// TwinCAT 3 PLC project PRG_B_BaseDecorator
// Title: B_BaseDecorate
// Company: RafalOS
// Author: Rafał Osajda
// ProjectVersion: 0.0.0.2
// ProgramVersion: 3.1.4024.0
// libraries:
//   B_Base, * (RafalOS)
//   Tc2_Standard, * (Beckhoff Automation GmbH)
//   Tc2_System, * (Beckhoff Automation GmbH)
//   Tc3_Module, * (Beckhoff Automation GmbH)
// project tree:
//   / PlcTask.TcTTO
//   POUs Compilation/ PRG_Compilation.TcPOU
//   POUs/A03_FB_BaseLoggerElementDecorator/ FB_BaseLoggerElementDecoratorParent.TcPOU, ITF_BaseLoggerElementDecoratorParent.TcIO
//   POUs/A04_FB_BaseComponentDecorator/ FB_BaseComponentDecoratorParent.TcPOU, ITF_BaseComponentDecoratorParent.TcIO
//   POUs/A05_FB_BaseControlElementDecorator/ FB_BaseControlElementDecoratorParent.TcPOU, ITF_BaseControlElementDecoratorParent.TcIO
//   POUs/A06_FB_BaseGroupElementDecorator/ FB_BaseGroupElementDecoratorParent.TcPOU, ITF_BaseGroupElementDecoratorParent.TcIO (not stored)
//   POUs/A07_FB_BaseTopElementDecorator/ FB_BaseTopElementDecoratorParent.TcPOU, ITF_BaseTopElementDecoratorParent.TcIO
// real-time tasks:
//   TASK PlcTask: cycle T#10ms, priority 20, ADS port 350

CONFIGURATION PRG_B_BaseDecorator
    RESOURCE PLC ON TwinCAT3
        TASK PlcTask(INTERVAL := T#10ms, PRIORITY := 20);
        PROGRAM PRG_Compilation WITH PlcTask : PRG_Compilation;
    END_RESOURCE
END_CONFIGURATION

// ---- POUs/A03_FB_BaseLoggerElementDecorator/ITF_BaseLoggerElementDecoratorParent.TcIO
INTERFACE ITF_BaseLoggerElementDecoratorParent EXTENDS ITF_BaseLoggerElement

END_INTERFACE

// ---- POUs/A04_FB_BaseComponentDecorator/ITF_BaseComponentDecoratorParent.TcIO
INTERFACE ITF_BaseComponentDecoratorParent EXTENDS ITF_BaseComponent

END_INTERFACE

// ---- POUs/A05_FB_BaseControlElementDecorator/ITF_BaseControlElementDecoratorParent.TcIO
INTERFACE ITF_BaseControlElementDecoratorParent EXTENDS ITF_BaseControlElement

END_INTERFACE

// ---- POUs/A07_FB_BaseTopElementDecorator/ITF_BaseTopElementDecoratorParent.TcIO
INTERFACE ITF_BaseTopElementDecoratorParent EXTENDS ITF_BaseTopElement

END_INTERFACE

// ---- POUs Compilation/PRG_Compilation.TcPOU
PROGRAM PRG_Compilation
VAR
	fbLoggerElement				: FB_BaseLoggerElement;
	fbLoggerElementDecorator	: FB_BaseLoggerElementDecoratorParent (fbToDecorate := fbLoggerElement);
END_VAR

END_PROGRAM

// ---- POUs/A03_FB_BaseLoggerElementDecorator/FB_BaseLoggerElementDecoratorParent.TcPOU
FUNCTION_BLOCK FB_BaseLoggerElementDecoratorParent IMPLEMENTS ITF_BaseLoggerElementDecoratorParent
VAR
	itfLoggerElement					: ITF_BaseLoggerElement;
END_VAR

(*			
	EVERDE sp. z o.o.
	Rafał Osajda		24.03.2025		TC 4024.66
	Definicja nowego zgłoszenia
*)
METHOD PUBLIC EventsDefinition : BOOL
EventsDefinition		:= THIS^.itfLoggerElement.EventsDefinition ();
END_METHOD

METHOD FB_init : BOOL
VAR_INPUT
	bInitRetains : BOOL; // if TRUE, the retain variables are initialized (warm start / cold start)
	bInCopyCode : BOOL;  // if TRUE, the instance afterwards gets moved into the copy code (online change)
	fbToDecorate		: ITF_DecoratedElement;
END_VAR
THIS^.itfLoggerElement	:= fbToDecorate.GetITFLoggerElement ();
END_METHOD

METHOD PUBLIC GetCode : STRING
VAR_INPUT
END_VAR
GetCode			:= THIS^.itfLoggerElement.GetCode ();
END_METHOD

METHOD PUBLIC GetID : UINT
VAR_INPUT
END_VAR
GetID		:= THIS^.itfLoggerElement.GetID ();
END_METHOD

METHOD PUBLIC GetIdentyfier : ST_BaseElementIdentifier
VAR_INPUT
END_VAR
GetIdentyfier		:= THIS^.itfLoggerElement.GetIdentyfier ();
END_METHOD

METHOD PUBLIC GetName : ST_BaseLabel
VAR_INPUT
END_VAR
GetName		:= THIS^.itfLoggerElement.GetName ();
END_METHOD

METHOD PUBLIC GetType : E_BaseElementType
VAR_INPUT
END_VAR
GetType		:= THIS^.itfLoggerElement.GetType ();
END_METHOD

METHOD PUBLIC SetCode
VAR_INPUT
	sCode							: STRING;
	sAdd							: STRING;
END_VAR
THIS^.itfLoggerElement.SetCode (sCode := sCode, sAdd := sAdd);
END_METHOD

(*			
	EVERDE sp. z o.o.
	Rafał Osajda		03.10.2025		TC 4024.66
	nadawanie unikalnych ID dla zdarzeń
*)
METHOD PUBLIC SetEventsIDs : UINT
VAR_INPUT
	uiNewID		: UINT;
END_VAR
SetEventsIDs		:= THIS^.itfLoggerElement.SetEventsIDs (uiNewID := uiNewID);
END_METHOD

METHOD PUBLIC SetID : UINT
VAR_INPUT
	uiID					: UINT;
END_VAR
SetID		:= THIS^.itfLoggerElement.SetID (uiID := uiID);
END_METHOD

METHOD PUBLIC SetName
VAR_INPUT
	stName				: ST_BaseLabel;
END_VAR
THIS^.itfLoggerElement.SetName (stName := stName);
END_METHOD

METHOD PUBLIC SetType
VAR_INPUT
	eType					: E_BaseElementType;
END_VAR
THIS^.itfLoggerElement.SetType (eType := eType);
END_METHOD

END_FUNCTION_BLOCK

// ---- POUs/A04_FB_BaseComponentDecorator/FB_BaseComponentDecoratorParent.TcPOU
FUNCTION_BLOCK FB_BaseComponentDecoratorParent EXTENDS FB_BaseLoggerElementDecoratorParent IMPLEMENTS ITF_BaseComponentDecoratorParent
VAR
	itfComponent				: ITF_BaseComponent;
END_VAR

(*			
	EVERDE sp. z o.o.
	Rafał Osajda		24.03.2025		TC 4024.66
	Definicja nowego zgłoszenia
*)
METHOD PUBLIC EventsDefinition : BOOL
EventsDefinition		:= THIS^.itfComponent.EventsDefinition ();
END_METHOD

(*			
	EVERDE sp. z o.o.
	Rafał Osajda		27.03.2025		TC 4024.66
	Obsluga bledow sprawdzanie czy jakis blad sie nei pojawil i ustawienie stanu lub wylaczenie
*)
METHOD PUBLIC ExecuteEveryCycle_Error
VAR_INPUT
END_VAR
THIS^.itfComponent.ExecuteEveryCycle_Error ();
END_METHOD

(*			
	EVERDE sp. z o.o.
	Rafał Osajda		27.03.2025		TC 4024.66
	Wywolanie co cykl operacji 
*)
METHOD PUBLIC ExecuteEveryCycle_Operation
VAR_INPUT
END_VAR
THIS^.itfComponent.ExecuteEveryCycle_Operation ();
END_METHOD

(*			
	EVERDE sp. z o.o.
	Rafał Osajda		27.03.2025		TC 4024.66
	Aktualizacja flag 
*)
METHOD PUBLIC ExecuteEveryCycle_Status
VAR_INST
END_VAR
THIS^.itfComponent.ExecuteEveryCycle_Status ();
END_METHOD

(*			
	EVERDE sp. z o.o.
	Rafał Osajda		27.03.2025		TC 4024.66
	Testowanie czy nei pojawil sie jakis rozkaz i uruchomienie odpowiednich operacji
*)
METHOD PUBLIC ExecuteEveryCycle_Test
VAR_INPUT
END_VAR
THIS^.itfComponent.ExecuteEveryCycle_Test ();
END_METHOD

METHOD FB_init : BOOL
VAR_INPUT
	bInitRetains : BOOL; // if TRUE, the retain variables are initialized (warm start / cold start)
	bInCopyCode : BOOL;  // if TRUE, the instance afterwards gets moved into the copy code (online change)
	fbToDecorate		: ITF_DecoratedElement;
END_VAR
THIS^.itfComponent		:= fbToDecorate.GetITFComponent ();
END_METHOD

(*			
	EVERDE sp. z o.o.
	Rafał Osajda		03.10.2025		TC 4024.66
	
*)
METHOD PUBLIC FirstCycle : BOOL
VAR_INPUT
END_VAR
FirstCycle				:= THIS^.itfComponent.FirstCycle ();
END_METHOD

METHOD PUBLIC GetCode : STRING
VAR_INPUT
END_VAR
GetCode			:= THIS^.itfComponent.GetCode ();
END_METHOD

METHOD PUBLIC GetID : UINT
VAR_INPUT
END_VAR
GetID		:= THIS^.itfComponent.GetID ();
END_METHOD

METHOD PUBLIC GetIdentyfier : ST_BaseElementIdentifier
VAR_INPUT
END_VAR
GetIdentyfier		:= THIS^.itfComponent.GetIdentyfier ();
END_METHOD

METHOD PUBLIC GetName : ST_BaseLabel
VAR_INPUT
END_VAR
GetName		:= THIS^.itfComponent.GetName ();
END_METHOD

METHOD PUBLIC GetType : E_BaseElementType
VAR_INPUT
END_VAR
GetType		:= THIS^.itfComponent.GetType ();
END_METHOD

METHOD PUBLIC IsValidCommonData : BOOL
VAR_INPUT
END_VAR
IsValidCommonData			:= THIS^.itfComponent.IsValidCommonData ();
END_METHOD

(*			
	EVERDE sp. z o.o.
	Rafał Osajda		07.10.2025		TC 4024.66
	Dodpisywanie się do listy logera
*)
METHOD PUBLIC JoinTheLogger : BOOL
VAR_INPUT
END_VAR
JoinTheLogger	:= THIS^.itfComponent.JoinTheLogger ();
END_METHOD

METHOD PUBLIC LinkCommonData : BOOL
VAR_INPUT
	stCommonData				: REFERENCE TO ST_BaseCommonData;
END_VAR
LinkCommonData			:= THIS^.itfComponent.LinkCommonData (stCommonData := stCommonData);
END_METHOD

(*			
	EVERDE sp. z o.o.
	Rafał Osajda		26.03.2025		TC 4024.66
	Zwraca wartość
*)
METHOD PUBLIC ParameterGetValue : REAL
VAR_INPUT
	uiNumber				: UINT;
END_VAR
ParameterGetValue			:= THIS^.itfComponent.ParameterGetValue (uiNumber := uiNumber);
END_METHOD

METHOD PUBLIC Reset : BOOL
VAR_INPUT
END_VAR
Reset	:= THIS^.itfComponent.Reset ();
END_METHOD

METHOD PUBLIC ResetGetBusy : BOOL
VAR_INPUT
END_VAR
ResetGetBusy		:= THIS^.itfComponent.ResetGetBusy ();
END_METHOD

METHOD PUBLIC ResetGetStatus : BOOL
VAR_INPUT
END_VAR
ResetGetStatus			:= THIS^.itfComponent.ResetGetStatus ();
END_METHOD

METHOD PUBLIC SetCode
VAR_INPUT
	sCode							: STRING;
	sAdd							: STRING;
END_VAR
THIS^.itfComponent.SetCode (sCode := sCode, sAdd := sAdd);
END_METHOD

(*			
	EVERDE sp. z o.o.
	Rafał Osajda		03.10.2025		TC 4024.66
	nadawanie unikalnych ID dla zdarzeń
*)
METHOD PUBLIC SetEventsIDs : UINT
VAR_INPUT
	uiNewID		: UINT;
END_VAR
SetEventsIDs		:= THIS^.itfComponent.SetEventsIDs (uiNewID := uiNewID);
END_METHOD

METHOD PUBLIC SetID : UINT
VAR_INPUT
	uiID					: UINT;
END_VAR
SetID		:= THIS^.itfComponent.SetID (uiID := uiID);
END_METHOD

METHOD PUBLIC SetName
VAR_INPUT
	stName				: ST_BaseLabel;
END_VAR
THIS^.itfComponent.SetName (stName := stName);
END_METHOD

METHOD PUBLIC SetType
VAR_INPUT
	eType					: E_BaseElementType;
END_VAR
THIS^.itfComponent.SetType (eType := eType);
END_METHOD

END_FUNCTION_BLOCK

// ---- POUs/A05_FB_BaseControlElementDecorator/FB_BaseControlElementDecoratorParent.TcPOU
FUNCTION_BLOCK FB_BaseControlElementDecoratorParent EXTENDS FB_BaseComponentDecoratorParent IMPLEMENTS ITF_BaseControlElementDecoratorParent
VAR
	itfControlElement				: ITF_BaseControlElement;
END_VAR

(*			
	EVERDE sp. z o.o.
	Rafał Osajda		24.03.2025		TC 4024.66
	Definicja nowego zgłoszenia
*)
METHOD PUBLIC EventsDefinition : BOOL
EventsDefinition		:= THIS^.itfControlElement.EventsDefinition ();
END_METHOD

(*			
	EVERDE sp. z o.o.
	Rafał Osajda		27.03.2025		TC 4024.66
	Obsluga bledow sprawdzanie czy jakis blad sie nei pojawil i ustawienie stanu lub wylaczenie
*)
METHOD PUBLIC ExecuteEveryCycle_Error
VAR_INPUT
END_VAR
THIS^.itfControlElement.ExecuteEveryCycle_Error ();
END_METHOD

(*			
	EVERDE sp. z o.o.
	Rafał Osajda		27.03.2025		TC 4024.66
	Wywolanie co cykl operacji 
*)
METHOD PUBLIC ExecuteEveryCycle_Operation
VAR_INPUT
END_VAR
THIS^.itfControlElement.ExecuteEveryCycle_Operation ();
END_METHOD

(*			
	EVERDE sp. z o.o.
	Rafał Osajda		27.03.2025		TC 4024.66
	Aktualizacja flag 
*)
METHOD PUBLIC ExecuteEveryCycle_Status
VAR_INST
END_VAR
THIS^.itfControlElement.ExecuteEveryCycle_Status ();
END_METHOD

(*			
	EVERDE sp. z o.o.
	Rafał Osajda		27.03.2025		TC 4024.66
	Testowanie czy nei pojawil sie jakis rozkaz i uruchomienie odpowiednich operacji
*)
METHOD PUBLIC ExecuteEveryCycle_Test
VAR_INPUT
END_VAR
THIS^.itfControlElement.ExecuteEveryCycle_Test ();
END_METHOD

METHOD FB_init : BOOL
VAR_INPUT
	bInitRetains : BOOL; // if TRUE, the retain variables are initialized (warm start / cold start)
	bInCopyCode : BOOL;  // if TRUE, the instance afterwards gets moved into the copy code (online change)
	fbToDecorate		: ITF_DecoratedElement;
END_VAR
THIS^.itfControlElement	:= fbToDecorate.GetITFControlElement ();
END_METHOD

(*			
	EVERDE sp. z o.o.
	Rafał Osajda		03.10.2025		TC 4024.66
	
*)
METHOD PUBLIC FirstCycle : BOOL
VAR_INPUT
END_VAR
FirstCycle				:= THIS^.itfControlElement.FirstCycle ();
END_METHOD

METHOD PUBLIC GetCode : STRING
VAR_INPUT
END_VAR
GetCode			:= THIS^.itfControlElement.GetCode ();
END_METHOD

(*			
	EVERDE sp. z o.o.
	Rafał Osajda		30.04.2025		TC 4024.66
	Zwraca czy element jest czymś zajety
*)
METHOD PUBLIC GetDoNothing : BOOL
GetDoNothing		:= THIS^.itfControlElement.GetDoNothing ();
END_METHOD

METHOD PUBLIC GetID : UINT
VAR_INPUT
END_VAR
GetID		:= THIS^.itfControlElement.GetID ();
END_METHOD

METHOD PUBLIC GetIdentyfier : ST_BaseElementIdentifier
VAR_INPUT
END_VAR
GetIdentyfier		:= THIS^.itfControlElement.GetIdentyfier ();
END_METHOD

METHOD PUBLIC GetName : ST_BaseLabel
VAR_INPUT
END_VAR
GetName		:= THIS^.itfControlElement.GetName ();
END_METHOD

(*			
	EVERDE sp. z o.o.
	Rafał Osajda		30.04.2025		TC 4024.66
	Zwraca czy element jest w pozycji 0 - referencyjnej
*)
METHOD PUBLIC GetPosition0 : BOOL
GetPosition0	:= THIS^.itfControlElement.GetPosition0 ();
END_METHOD

METHOD PUBLIC GetType : E_BaseElementType
VAR_INPUT
END_VAR
GetType		:= THIS^.itfControlElement.GetType ();
END_METHOD

(*			
	EVERDE sp. z o.o.
	Rafał Osajda		31.03.2025		TC 4024.66
	Flaga że w tej sesji pracy maszyny element został już wybazowany
*)
METHOD PUBLIC HomingGetDone : BOOL
VAR_INPUT
END_VAR
HomingGetDone	:= THIS^.itfControlElement.HomingGetDone ();
END_METHOD

(*			
	EVERDE sp. z o.o.
	Rafał Osajda		11.04.2025		TC 4024.66
	Zwraca czy bazowanie jest potrzebne
*)
METHOD PUBLIC HomingGetIsNeeded : BOOL
VAR_INPUT
END_VAR
HomingGetIsNeeded	:= THIS^.itfControlElement.HomingGetIsNeeded ();
END_METHOD

(*			
	EVERDE sp. z o.o.
	Rafał Osajda		27.05.2025		TC 4024.66
	Uruchomienie metody bazowania
*)
METHOD PUBLIC HomingStart
VAR_INPUT
END_VAR
THIS^.itfControlElement.HomingStart ();
END_METHOD

METHOD PUBLIC IsValidCommonData : BOOL
VAR_INPUT
END_VAR
IsValidCommonData			:= THIS^.itfControlElement.IsValidCommonData ();
END_METHOD

(*			
	EVERDE sp. z o.o.
	Rafał Osajda		07.10.2025		TC 4024.66
	Dodpisywanie się do listy logera
*)
METHOD PUBLIC JoinTheLogger : BOOL
VAR_INPUT
END_VAR
JoinTheLogger	:= THIS^.itfControlElement.JoinTheLogger ();
END_METHOD

METHOD PUBLIC LinkCommonData : BOOL
VAR_INPUT
	stCommonData				: REFERENCE TO ST_BaseCommonData;
END_VAR
LinkCommonData			:= THIS^.itfControlElement.LinkCommonData (stCommonData := stCommonData);
END_METHOD

METHOD PUBLIC LinkSS1 : BOOL
VAR_INPUT
	fbSS1			: ITF_BaseFlagGet;
END_VAR
LinkSS1		:= THIS^.itfControlElement.LinkSS1 (fbSS1 := fbSS1);
END_METHOD

METHOD PUBLIC LinkSTO : BOOL
VAR_INPUT
	fbSTO			: ITF_BaseFlagGet;
END_VAR
LinkSTO		:= THIS^.itfControlElement.LinkSTO (fbSTO := fbSTO);
END_METHOD

(*			
	EVERDE sp. z o.o.
	Rafał Osajda		31.03.2025		TC 4024.66
	Zwraca status zasilania	
*)
METHOD PUBLIC PowerGetStatus : BOOL
VAR_INPUT
END_VAR
PowerGetStatus		:= THIS^.itfControlElement.PowerGetStatus ();
END_METHOD

(*			
	EVERDE sp. z o.o.
	Rafał Osajda		31.03.2025		TC 4024.66
	Wyłączenie zasilania
*)
METHOD PUBLIC PowerTurnOff : BOOL
VAR_INPUT
END_VAR
PowerTurnOff		:= THIS^.itfControlElement.PowerTurnOff ();
END_METHOD

(*			
	EVERDE sp. z o.o.
	Rafał Osajda		31.03.2025		TC 4024.66
	Uruchomienie zasialania
*)
METHOD PUBLIC PowerTurnOn
VAR_INPUT
END_VAR
THIS^.itfControlElement.PowerTurnOn ();
END_METHOD

METHOD PUBLIC Reset : BOOL
VAR_INPUT
END_VAR
Reset	:= THIS^.itfControlElement.Reset ();
END_METHOD

METHOD PUBLIC ResetGetBusy : BOOL
VAR_INPUT
END_VAR
ResetGetBusy		:= THIS^.itfControlElement.ResetGetBusy ();
END_METHOD

METHOD PUBLIC ResetGetStatus : BOOL
VAR_INPUT
END_VAR
ResetGetStatus			:= THIS^.itfControlElement.ResetGetStatus ();
END_METHOD

METHOD PUBLIC SetCode
VAR_INPUT
	sCode							: STRING;
	sAdd							: STRING;
END_VAR
THIS^.itfControlElement.SetCode (sCode := sCode, sAdd := sAdd);
END_METHOD

(*			
	EVERDE sp. z o.o.
	Rafał Osajda		03.10.2025		TC 4024.66
	nadawanie unikalnych ID dla zdarzeń
*)
METHOD PUBLIC SetEventsIDs : UINT
VAR_INPUT
	uiNewID		: UINT;
END_VAR
SetEventsIDs		:= THIS^.itfControlElement.SetEventsIDs (uiNewID := uiNewID);
END_METHOD

METHOD PUBLIC SetID : UINT
VAR_INPUT
	uiID					: UINT;
END_VAR
SetID		:= THIS^.itfControlElement.SetID (uiID := uiID);
END_METHOD

METHOD PUBLIC SetName
VAR_INPUT
	stName				: ST_BaseLabel;
END_VAR
THIS^.itfControlElement.SetName (stName := stName);
END_METHOD

METHOD PUBLIC SetType
VAR_INPUT
	eType					: E_BaseElementType;
END_VAR
THIS^.itfControlElement.SetType (eType := eType);
END_METHOD

END_FUNCTION_BLOCK

// ---- POUs/A06_FB_BaseGroupElementDecorator/FB_BaseGroupElementDecoratorParent.TcPOU
FUNCTION_BLOCK FB_BaseGroupElementDecoratorParent EXTENDS FB_BaseControlElementDecoratorParent IMPLEMENTS ITF_BaseGroupElementDecoratorParent
VAR
	itfGroupElement				: ITF_BaseGroupElement;
END_VAR

(*			
	EVERDE sp. z o.o.
	Rafał Osajda		24.03.2025		TC 4024.66
	Definicja nowego zgłoszenia
*)
METHOD PUBLIC EventsDefinition : BOOL
EventsDefinition		:= THIS^.itfGroupElement.EventsDefinition ();
END_METHOD

(*			
	EVERDE sp. z o.o.
	Rafał Osajda		27.03.2025		TC 4024.66
	Obsluga bledow sprawdzanie czy jakis blad sie nei pojawil i ustawienie stanu lub wylaczenie
*)
METHOD PUBLIC ExecuteEveryCycle_Error
VAR_INPUT
END_VAR
THIS^.itfGroupElement.ExecuteEveryCycle_Error ();
END_METHOD

(*			
	EVERDE sp. z o.o.
	Rafał Osajda		27.03.2025		TC 4024.66
	Wywolanie co cykl operacji 
*)
METHOD PUBLIC ExecuteEveryCycle_Operation
VAR_INPUT
END_VAR
THIS^.itfGroupElement.ExecuteEveryCycle_Operation ();
END_METHOD

(*			
	EVERDE sp. z o.o.
	Rafał Osajda		27.03.2025		TC 4024.66
	Aktualizacja flag 
*)
METHOD PUBLIC ExecuteEveryCycle_Status
VAR_INST
END_VAR
THIS^.itfGroupElement.ExecuteEveryCycle_Status ();
END_METHOD

(*			
	EVERDE sp. z o.o.
	Rafał Osajda		27.03.2025		TC 4024.66
	Testowanie czy nei pojawil sie jakis rozkaz i uruchomienie odpowiednich operacji
*)
METHOD PUBLIC ExecuteEveryCycle_Test
VAR_INPUT
END_VAR
THIS^.itfGroupElement.ExecuteEveryCycle_Test ();
END_METHOD

METHOD FB_init : BOOL
VAR_INPUT
	bInitRetains : BOOL; // if TRUE, the retain variables are initialized (warm start / cold start)
	bInCopyCode : BOOL;  // if TRUE, the instance afterwards gets moved into the copy code (online change)
	fbToDecorate		: ITF_DecoratedElement;
END_VAR
THIS^.itfGroupElement	:= fbToDecorate.GetITFGroupElement ();
END_METHOD

(*			
	EVERDE sp. z o.o.
	Rafał Osajda		03.10.2025		TC 4024.66
	
*)
METHOD PUBLIC FirstCycle : BOOL
VAR_INPUT
END_VAR
FirstCycle				:= THIS^.itfGroupElement.FirstCycle ();
END_METHOD

METHOD PUBLIC GetCode : STRING
VAR_INPUT
END_VAR
GetCode			:= THIS^.itfGroupElement.GetCode ();
END_METHOD

(*			
	EVERDE sp. z o.o.
	Rafał Osajda		30.04.2025		TC 4024.66
	Zwraca czy element jest czymś zajety
*)
METHOD PUBLIC GetDoNothing : BOOL
GetDoNothing		:= THIS^.itfGroupElement.GetDoNothing ();
END_METHOD

METHOD PUBLIC GetID : UINT
VAR_INPUT
END_VAR
GetID		:= THIS^.itfGroupElement.GetID ();
END_METHOD

METHOD PUBLIC GetIdentyfier : ST_BaseElementIdentifier
VAR_INPUT
END_VAR
GetIdentyfier		:= THIS^.itfGroupElement.GetIdentyfier ();
END_METHOD

METHOD PUBLIC GetName : ST_BaseLabel
VAR_INPUT
END_VAR
GetName		:= THIS^.itfGroupElement.GetName ();
END_METHOD

(*			
	EVERDE sp. z o.o.
	Rafał Osajda		30.04.2025		TC 4024.66
	Zwraca czy element jest w pozycji 0 - referencyjnej
*)
METHOD PUBLIC GetPosition0 : BOOL
GetPosition0	:= THIS^.itfGroupElement.GetPosition0 ();
END_METHOD

METHOD PUBLIC GetType : E_BaseElementType
VAR_INPUT
END_VAR
GetType		:= THIS^.itfGroupElement.GetType ();
END_METHOD

(*			
	EVERDE sp. z o.o.
	Rafał Osajda		31.03.2025		TC 4024.66
	Flaga że w tej sesji pracy maszyny element został już wybazowany
*)
METHOD PUBLIC HomingGetDone : BOOL
VAR_INPUT
END_VAR
HomingGetDone	:= THIS^.itfGroupElement.HomingGetDone ();
END_METHOD

(*			
	EVERDE sp. z o.o.
	Rafał Osajda		11.04.2025		TC 4024.66
	Zwraca czy bazowanie jest potrzebne
*)
METHOD PUBLIC HomingGetIsNeeded : BOOL
VAR_INPUT
END_VAR
HomingGetIsNeeded	:= THIS^.itfGroupElement.HomingGetIsNeeded ();
END_METHOD

(*			
	EVERDE sp. z o.o.
	Rafał Osajda		27.05.2025		TC 4024.66
	Uruchomienie metody bazowania
*)
METHOD PUBLIC HomingStart
VAR_INPUT
END_VAR
THIS^.itfGroupElement.HomingStart ();
END_METHOD

METHOD PUBLIC IsValidCommonData : BOOL
VAR_INPUT
END_VAR
IsValidCommonData			:= THIS^.itfGroupElement.IsValidCommonData ();
END_METHOD

(*			
	EVERDE sp. z o.o.
	Rafał Osajda		07.10.2025		TC 4024.66
	Dodpisywanie się do listy logera
*)
METHOD PUBLIC JoinTheLogger : BOOL
VAR_INPUT
END_VAR
JoinTheLogger	:= THIS^.itfGroupElement.JoinTheLogger ();
END_METHOD

METHOD PUBLIC LinkCommonData : BOOL
VAR_INPUT
	stCommonData				: REFERENCE TO ST_BaseCommonData;
END_VAR
LinkCommonData			:= THIS^.itfGroupElement.LinkCommonData (stCommonData := stCommonData);
END_METHOD

METHOD PUBLIC LinkSS1 : BOOL
VAR_INPUT
	fbSS1			: ITF_BaseFlagGet;
END_VAR
LinkSS1		:= THIS^.itfGroupElement.LinkSS1 (fbSS1 := fbSS1);
END_METHOD

METHOD PUBLIC LinkSTO : BOOL
VAR_INPUT
	fbSTO			: ITF_BaseFlagGet;
END_VAR
LinkSTO		:= THIS^.itfGroupElement.LinkSTO (fbSTO := fbSTO);
END_METHOD

(*			
	EVERDE sp. z o.o.
	Rafał Osajda		31.03.2025		TC 4024.66
	Zwraca status zasilania	
*)
METHOD PUBLIC PowerGetStatus : BOOL
VAR_INPUT
END_VAR
PowerGetStatus		:= THIS^.itfGroupElement.PowerGetStatus ();
END_METHOD

(*			
	EVERDE sp. z o.o.
	Rafał Osajda		31.03.2025		TC 4024.66
	Wyłączenie zasilania
*)
METHOD PUBLIC PowerTurnOff : BOOL
VAR_INPUT
END_VAR
PowerTurnOff		:= THIS^.itfGroupElement.PowerTurnOff ();
END_METHOD

(*			
	EVERDE sp. z o.o.
	Rafał Osajda		31.03.2025		TC 4024.66
	Uruchomienie zasialania
*)
METHOD PUBLIC PowerTurnOn
VAR_INPUT
END_VAR
THIS^.itfGroupElement.PowerTurnOn ();
END_METHOD

METHOD PUBLIC Reset : BOOL
VAR_INPUT
END_VAR
Reset	:= THIS^.itfGroupElement.Reset ();
END_METHOD

METHOD PUBLIC ResetGetBusy : BOOL
VAR_INPUT
END_VAR
ResetGetBusy		:= THIS^.itfGroupElement.ResetGetBusy ();
END_METHOD

METHOD PUBLIC ResetGetStatus : BOOL
VAR_INPUT
END_VAR
ResetGetStatus			:= THIS^.itfGroupElement.ResetGetStatus ();
END_METHOD

METHOD PUBLIC SetCode
VAR_INPUT
	sCode							: STRING;
	sAdd							: STRING;
END_VAR
THIS^.itfGroupElement.SetCode (sCode := sCode, sAdd := sAdd);
END_METHOD

(*			
	EVERDE sp. z o.o.
	Rafał Osajda		03.10.2025		TC 4024.66
	nadawanie unikalnych ID dla zdarzeń
*)
METHOD PUBLIC SetEventsIDs : UINT
VAR_INPUT
	uiNewID		: UINT;
END_VAR
SetEventsIDs		:= THIS^.itfGroupElement.SetEventsIDs (uiNewID := uiNewID);
END_METHOD

METHOD PUBLIC SetID : UINT
VAR_INPUT
	uiID					: UINT;
END_VAR
SetID		:= THIS^.itfGroupElement.SetID (uiID := uiID);
END_METHOD

METHOD PUBLIC SetName
VAR_INPUT
	stName				: ST_BaseLabel;
END_VAR
THIS^.itfGroupElement.SetName (stName := stName);
END_METHOD

METHOD PUBLIC SetType
VAR_INPUT
	eType					: E_BaseElementType;
END_VAR
THIS^.itfGroupElement.SetType (eType := eType);
END_METHOD

END_FUNCTION_BLOCK

// ---- POUs/A07_FB_BaseTopElementDecorator/FB_BaseTopElementDecoratorParent.TcPOU
FUNCTION_BLOCK FB_BaseTopElementDecoratorParent EXTENDS FB_BaseGroupElementDecoratorParent IMPLEMENTS ITF_BaseTopElementDecoratorParent
VAR
	itfTopElement				: ITF_BaseTopElement;
END_VAR

(*			
	EVERDE sp. z o.o.
	Rafał Osajda		24.03.2025		TC 4024.66
	Definicja nowego zgłoszenia
*)
METHOD PUBLIC EventsDefinition : BOOL
EventsDefinition		:= THIS^.itfTopElement.EventsDefinition ();
END_METHOD

(*			
	EVERDE sp. z o.o.
	Rafał Osajda		27.03.2025		TC 4024.66
	Obsluga bledow sprawdzanie czy jakis blad sie nei pojawil i ustawienie stanu lub wylaczenie
*)
METHOD PUBLIC ExecuteEveryCycle_Error
VAR_INPUT
END_VAR
THIS^.itfTopElement.ExecuteEveryCycle_Error ();
END_METHOD

(*			
	EVERDE sp. z o.o.
	Rafał Osajda		27.03.2025		TC 4024.66
	Wywolanie co cykl operacji 
*)
METHOD PUBLIC ExecuteEveryCycle_Operation
VAR_INPUT
END_VAR
THIS^.itfTopElement.ExecuteEveryCycle_Operation ();
END_METHOD

(*			
	EVERDE sp. z o.o.
	Rafał Osajda		27.03.2025		TC 4024.66
	Aktualizacja flag 
*)
METHOD PUBLIC ExecuteEveryCycle_Status
VAR_INST
END_VAR
THIS^.itfTopElement.ExecuteEveryCycle_Status ();
END_METHOD

(*			
	EVERDE sp. z o.o.
	Rafał Osajda		27.03.2025		TC 4024.66
	Testowanie czy nei pojawil sie jakis rozkaz i uruchomienie odpowiednich operacji
*)
METHOD PUBLIC ExecuteEveryCycle_Test
VAR_INPUT
END_VAR
THIS^.itfTopElement.ExecuteEveryCycle_Test ();
END_METHOD

METHOD FB_init : BOOL
VAR_INPUT
	bInitRetains : BOOL; // if TRUE, the retain variables are initialized (warm start / cold start)
	bInCopyCode : BOOL;  // if TRUE, the instance afterwards gets moved into the copy code (online change)
	fbToDecorate		: ITF_DecoratedElement;
END_VAR
THIS^.itfTopElement	:= fbToDecorate.GetITFTopElement ();
END_METHOD

(*			
	EVERDE sp. z o.o.
	Rafał Osajda		03.10.2025		TC 4024.66
	
*)
METHOD PUBLIC FirstCycle : BOOL
VAR_INPUT
END_VAR
FirstCycle				:= THIS^.itfTopElement.FirstCycle ();
END_METHOD

METHOD PUBLIC GetCode : STRING
VAR_INPUT
END_VAR
GetCode			:= THIS^.itfTopElement.GetCode ();
END_METHOD

(*			
	EVERDE sp. z o.o.
	Rafał Osajda		30.04.2025		TC 4024.66
	Zwraca czy element jest czymś zajety
*)
METHOD PUBLIC GetDoNothing : BOOL
GetDoNothing		:= THIS^.itfTopElement.GetDoNothing ();
END_METHOD

METHOD PUBLIC GetID : UINT
VAR_INPUT
END_VAR
GetID		:= THIS^.itfTopElement.GetID ();
END_METHOD

METHOD PUBLIC GetIdentyfier : ST_BaseElementIdentifier
VAR_INPUT
END_VAR
GetIdentyfier		:= THIS^.itfTopElement.GetIdentyfier ();
END_METHOD

METHOD PUBLIC GetName : ST_BaseLabel
VAR_INPUT
END_VAR
GetName		:= THIS^.itfTopElement.GetName ();
END_METHOD

(*			
	EVERDE sp. z o.o.
	Rafał Osajda		30.04.2025		TC 4024.66
	Zwraca czy element jest w pozycji 0 - referencyjnej
*)
METHOD PUBLIC GetPosition0 : BOOL
GetPosition0	:= THIS^.itfTopElement.GetPosition0 ();
END_METHOD

METHOD PUBLIC GetType : E_BaseElementType
VAR_INPUT
END_VAR
GetType		:= THIS^.itfTopElement.GetType ();
END_METHOD

(*			
	EVERDE sp. z o.o.
	Rafał Osajda		31.03.2025		TC 4024.66
	Flaga że w tej sesji pracy maszyny element został już wybazowany
*)
METHOD PUBLIC HomingGetDone : BOOL
VAR_INPUT
END_VAR
HomingGetDone	:= THIS^.itfTopElement.HomingGetDone ();
END_METHOD

(*			
	EVERDE sp. z o.o.
	Rafał Osajda		11.04.2025		TC 4024.66
	Zwraca czy bazowanie jest potrzebne
*)
METHOD PUBLIC HomingGetIsNeeded : BOOL
VAR_INPUT
END_VAR
HomingGetIsNeeded	:= THIS^.itfTopElement.HomingGetIsNeeded ();
END_METHOD

(*			
	EVERDE sp. z o.o.
	Rafał Osajda		27.05.2025		TC 4024.66
	Uruchomienie metody bazowania
*)
METHOD PUBLIC HomingStart
VAR_INPUT
END_VAR
THIS^.itfTopElement.HomingStart ();
END_METHOD

METHOD PUBLIC IsValidCommonData : BOOL
VAR_INPUT
END_VAR
IsValidCommonData			:= THIS^.itfTopElement.IsValidCommonData ();
END_METHOD

(*			
	EVERDE sp. z o.o.
	Rafał Osajda		07.10.2025		TC 4024.66
	Dodpisywanie się do listy logera
*)
METHOD PUBLIC JoinTheLogger : BOOL
VAR_INPUT
END_VAR
JoinTheLogger	:= THIS^.itfTopElement.JoinTheLogger ();
END_METHOD

METHOD PUBLIC LinkCommonData : BOOL
VAR_INPUT
	stCommonData				: REFERENCE TO ST_BaseCommonData;
END_VAR
LinkCommonData			:= THIS^.itfTopElement.LinkCommonData (stCommonData := stCommonData);
END_METHOD

METHOD PUBLIC LinkSS1 : BOOL
VAR_INPUT
	fbSS1			: ITF_BaseFlagGet;
END_VAR
LinkSS1		:= THIS^.itfTopElement.LinkSS1 (fbSS1 := fbSS1);
END_METHOD

METHOD PUBLIC LinkSTO : BOOL
VAR_INPUT
	fbSTO			: ITF_BaseFlagGet;
END_VAR
LinkSTO		:= THIS^.itfTopElement.LinkSTO (fbSTO := fbSTO);
END_METHOD

(*			
	EVERDE sp. z o.o.
	Rafał Osajda		31.03.2025		TC 4024.66
	Zwraca status zasilania	
*)
METHOD PUBLIC PowerGetStatus : BOOL
VAR_INPUT
END_VAR
PowerGetStatus		:= THIS^.itfTopElement.PowerGetStatus ();
END_METHOD

(*			
	EVERDE sp. z o.o.
	Rafał Osajda		31.03.2025		TC 4024.66
	Wyłączenie zasilania
*)
METHOD PUBLIC PowerTurnOff : BOOL
VAR_INPUT
END_VAR
PowerTurnOff		:= THIS^.itfTopElement.PowerTurnOff ();
END_METHOD

(*			
	EVERDE sp. z o.o.
	Rafał Osajda		31.03.2025		TC 4024.66
	Uruchomienie zasialania
*)
METHOD PUBLIC PowerTurnOn
VAR_INPUT
END_VAR
THIS^.itfTopElement.PowerTurnOn ();
END_METHOD

METHOD PUBLIC Reset : BOOL
VAR_INPUT
END_VAR
Reset	:= THIS^.itfTopElement.Reset ();
END_METHOD

METHOD PUBLIC ResetGetBusy : BOOL
VAR_INPUT
END_VAR
ResetGetBusy		:= THIS^.itfTopElement.ResetGetBusy ();
END_METHOD

METHOD PUBLIC ResetGetStatus : BOOL
VAR_INPUT
END_VAR
ResetGetStatus			:= THIS^.itfTopElement.ResetGetStatus ();
END_METHOD

METHOD PUBLIC SetCode
VAR_INPUT
	sCode							: STRING;
	sAdd							: STRING;
END_VAR
THIS^.itfTopElement.SetCode (sCode := sCode, sAdd := sAdd);
END_METHOD

(*			
	EVERDE sp. z o.o.
	Rafał Osajda		03.10.2025		TC 4024.66
	nadawanie unikalnych ID dla zdarzeń
*)
METHOD PUBLIC SetEventsIDs : UINT
VAR_INPUT
	uiNewID		: UINT;
END_VAR
SetEventsIDs		:= THIS^.itfTopElement.SetEventsIDs (uiNewID := uiNewID);
END_METHOD

METHOD PUBLIC SetID : UINT
VAR_INPUT
	uiID					: UINT;
END_VAR
SetID		:= THIS^.itfTopElement.SetID (uiID := uiID);
END_METHOD

METHOD PUBLIC SetName
VAR_INPUT
	stName				: ST_BaseLabel;
END_VAR
THIS^.itfTopElement.SetName (stName := stName);
END_METHOD

METHOD PUBLIC SetType
VAR_INPUT
	eType					: E_BaseElementType;
END_VAR
THIS^.itfTopElement.SetType (eType := eType);
END_METHOD

END_FUNCTION_BLOCK
